// TIA Portal V19 export
TYPE "ValveMachine_Wng"
// stored: Access Published
   STRUCT
      NotAutReady : Bool;
      PressureRunning_Timeout : Bool;
      Rest_MissingExtEnable : Bool;
      Work_MissingExtEnable : Bool;
      Missing_Rest_Ls_ON : Array[1..8] of Bool;
      Missing_Work_Ls_ON : Array[1..8] of Bool;
   END_STRUCT;
END_TYPE
